// TIA Portal V16 export
// export: Created 2021-12-01T21:20:16.7242301Z, ExportSetting WithDefaults, DisplayName Totally Integrated Automation Portal, DisplayVersion V16 Update 4, DisplayName TIA Portal Version Control Interface, DisplayVersion V16 Update 2, DisplayName TIA Portal Openness, DisplayVersion V16 Update 4, DisplayName SINAMICS Startdrive Advanced, DisplayVersion V16 Update 5, DisplayName SINAMICS Startdrive G130, G150, S120, S150, SINAMICS MV, S210, DisplayVersion V16 Update 5, DisplayName SINAMICS Startdrive G110M, G120, G120C, G120D, G120P, G115D, DisplayVersion V16 Update 5, DisplayName STEP 7 Professional, DisplayVersion V16 Update 4, DisplayName STEP 7 Safety, DisplayVersion V16, DisplayName WinCC Advanced, DisplayVersion V16 Update 4
FUNCTION "ST00270_FC" : Void   // FC157, LAD
TITLE = ST00270
{ S7_Optimized_Access := 'TRUE' }
VERSION : 0.1
// stored: AutoNumber true, IsIECCheckEnabled false, SetENOAutomatically false, UDAEnableTagReadback false
   VAR_IN_OUT
      OPMODE : "OPMODE_OUT_UDT";
      HMI_EXTENSION : "HMI_EXTENSION_PANEL_UDT";
   END_VAR
BEGIN

REGION Network 1: Alarm
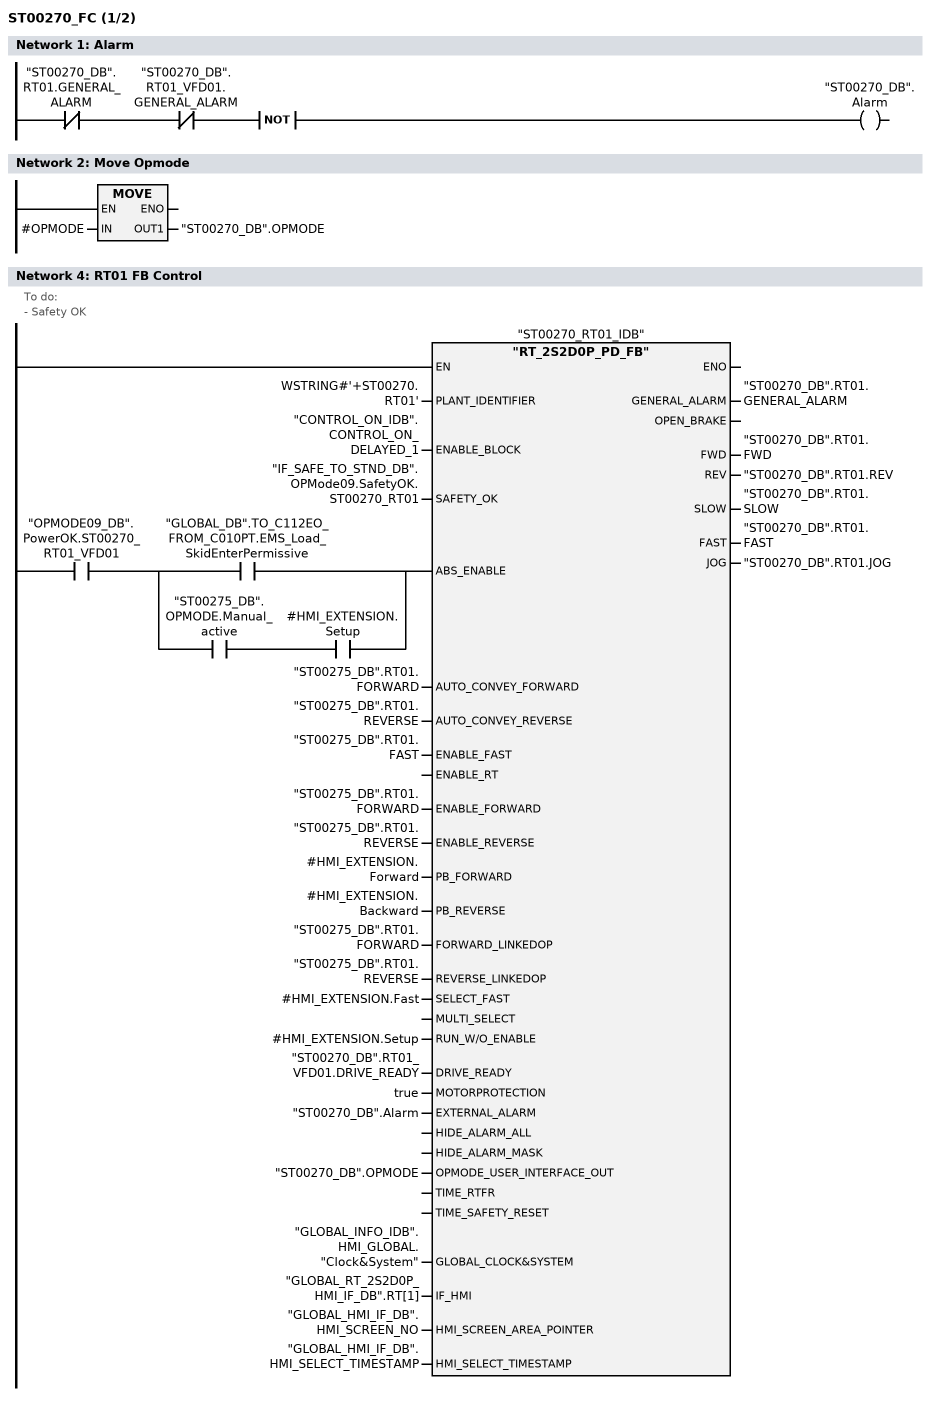
   RUNG wire#powerrail
      I_Contact( "ST00270_DB".RT01.GENERAL_ALARM )
      I_Contact( "ST00270_DB".RT01_VFD01.GENERAL_ALARM )
      Not()
      Coil( "ST00270_DB".Alarm )
   END_RUNG
   // the same network as SCL:
   "ST00270_DB".Alarm := NOT (NOT "ST00270_DB".RT01.GENERAL_ALARM AND NOT "ST00270_DB".RT01_VFD01.GENERAL_ALARM);
END_REGION

REGION Network 2: Move Opmode
   RUNG wire#powerrail
      Move(in := #OPMODE, out1 => "ST00270_DB".OPMODE)
   END_RUNG
   // the same network as SCL:
   "ST00270_DB".OPMODE := #OPMODE;
END_REGION

REGION Network 3: *******************RT01 Control*******************
END_REGION

REGION Network 4: RT01 FB Control
   // To do:
   // 										- Safety OK
   RUNG wire#powerrail
      "ST00270_RT01_IDB"(ABS_ENABLE := wire#w2, PLANT_IDENTIFIER := WSTRING#'+ST00270.RT01', ENABLE_BLOCK := "CONTROL_ON_IDB".CONTROL_ON_DELAYED_1, SAFETY_OK := "IF_SAFE_TO_STND_DB".OPMode09.SafetyOK.ST00270_RT01, AUTO_CONVEY_FORWARD := "ST00275_DB".RT01.FORWARD, AUTO_CONVEY_REVERSE := "ST00275_DB".RT01.REVERSE, ENABLE_FAST := "ST00275_DB".RT01.FAST, ENABLE_RT :=, ENABLE_FORWARD := "ST00275_DB".RT01.FORWARD, ENABLE_REVERSE := "ST00275_DB".RT01.REVERSE, PB_FORWARD := #HMI_EXTENSION.Forward, PB_REVERSE := #HMI_EXTENSION.Backward, FORWARD_LINKEDOP := "ST00275_DB".RT01.FORWARD, REVERSE_LINKEDOP := "ST00275_DB".RT01.REVERSE, SELECT_FAST := #HMI_EXTENSION.Fast, MULTI_SELECT :=, "RUN_W/O_ENABLE" := #HMI_EXTENSION.Setup, DRIVE_READY := "ST00270_DB".RT01_VFD01.DRIVE_READY, MOTORPROTECTION := true, EXTERNAL_ALARM := "ST00270_DB".Alarm, HIDE_ALARM_ALL :=, HIDE_ALARM_MASK :=, OPMODE_USER_INTERFACE_OUT := "ST00270_DB".OPMODE, TIME_RTFR :=, TIME_SAFETY_RESET :=, "GLOBAL_CLOCK&SYSTEM" := "GLOBAL_INFO_IDB".HMI_GLOBAL."Clock&System", IF_HMI := "GLOBAL_RT_2S2D0P_HMI_IF_DB".RT[1], HMI_SCREEN_AREA_POINTER := "GLOBAL_HMI_IF_DB".HMI_SCREEN_NO, HMI_SELECT_TIMESTAMP := "GLOBAL_HMI_IF_DB".HMI_SELECT_TIMESTAMP, GENERAL_ALARM => "ST00270_DB".RT01.GENERAL_ALARM, OPEN_BRAKE =>, FWD => "ST00270_DB".RT01.FWD, REV => "ST00270_DB".RT01.REV, SLOW => "ST00270_DB".RT01.SLOW, FAST => "ST00270_DB".RT01.FAST, JOG => "ST00270_DB".RT01.JOG)
   END_RUNG
   RUNG wire#powerrail
      Contact( "OPMODE09_DB".PowerOK.ST00270_RT01_VFD01 )
      wire#w1
      Contact( "GLOBAL_DB".TO_C112EO_FROM_C010PT.EMS_Load_SkidEnterPermissive )
   END_RUNG wire#w2
   RUNG wire#w1
      Contact( "ST00275_DB".OPMODE.Manual_active )
      Contact( #HMI_EXTENSION.Setup )
   END_RUNG wire#w2
   // the same network as SCL:
   "ST00270_RT01_IDB"(PLANT_IDENTIFIER := WSTRING#'+ST00270.RT01',   // "RT_2S2D0P_PD_FB"
                      ENABLE_BLOCK := "CONTROL_ON_IDB".CONTROL_ON_DELAYED_1,
                      SAFETY_OK := "IF_SAFE_TO_STND_DB".OPMode09.SafetyOK.ST00270_RT01,
                      ABS_ENABLE := "OPMODE09_DB".PowerOK.ST00270_RT01_VFD01 AND ("GLOBAL_DB".TO_C112EO_FROM_C010PT.EMS_Load_SkidEnterPermissive OR ("ST00275_DB".OPMODE.Manual_active AND #HMI_EXTENSION.Setup)),
                      AUTO_CONVEY_FORWARD := "ST00275_DB".RT01.FORWARD,
                      AUTO_CONVEY_REVERSE := "ST00275_DB".RT01.REVERSE,
                      ENABLE_FAST := "ST00275_DB".RT01.FAST,
                      ENABLE_FORWARD := "ST00275_DB".RT01.FORWARD,
                      ENABLE_REVERSE := "ST00275_DB".RT01.REVERSE,
                      PB_FORWARD := #HMI_EXTENSION.Forward,
                      PB_REVERSE := #HMI_EXTENSION.Backward,
                      FORWARD_LINKEDOP := "ST00275_DB".RT01.FORWARD,
                      REVERSE_LINKEDOP := "ST00275_DB".RT01.REVERSE,
                      SELECT_FAST := #HMI_EXTENSION.Fast,
                      "RUN_W/O_ENABLE" := #HMI_EXTENSION.Setup,
                      DRIVE_READY := "ST00270_DB".RT01_VFD01.DRIVE_READY,
                      MOTORPROTECTION := true,
                      EXTERNAL_ALARM := "ST00270_DB".Alarm,
                      OPMODE_USER_INTERFACE_OUT := "ST00270_DB".OPMODE,
                      "GLOBAL_CLOCK&SYSTEM" := "GLOBAL_INFO_IDB".HMI_GLOBAL."Clock&System",
                      IF_HMI := "GLOBAL_RT_2S2D0P_HMI_IF_DB".RT[1],
                      HMI_SCREEN_AREA_POINTER := "GLOBAL_HMI_IF_DB".HMI_SCREEN_NO,
                      HMI_SELECT_TIMESTAMP := "GLOBAL_HMI_IF_DB".HMI_SELECT_TIMESTAMP,
                      GENERAL_ALARM => "ST00270_DB".RT01.GENERAL_ALARM,
                      FWD => "ST00270_DB".RT01.FWD,
                      REV => "ST00270_DB".RT01.REV,
                      SLOW => "ST00270_DB".RT01.SLOW,
                      FAST => "ST00270_DB".RT01.FAST,
                      JOG => "ST00270_DB".RT01.JOG);
END_REGION

REGION Network 5: RT01 Speed
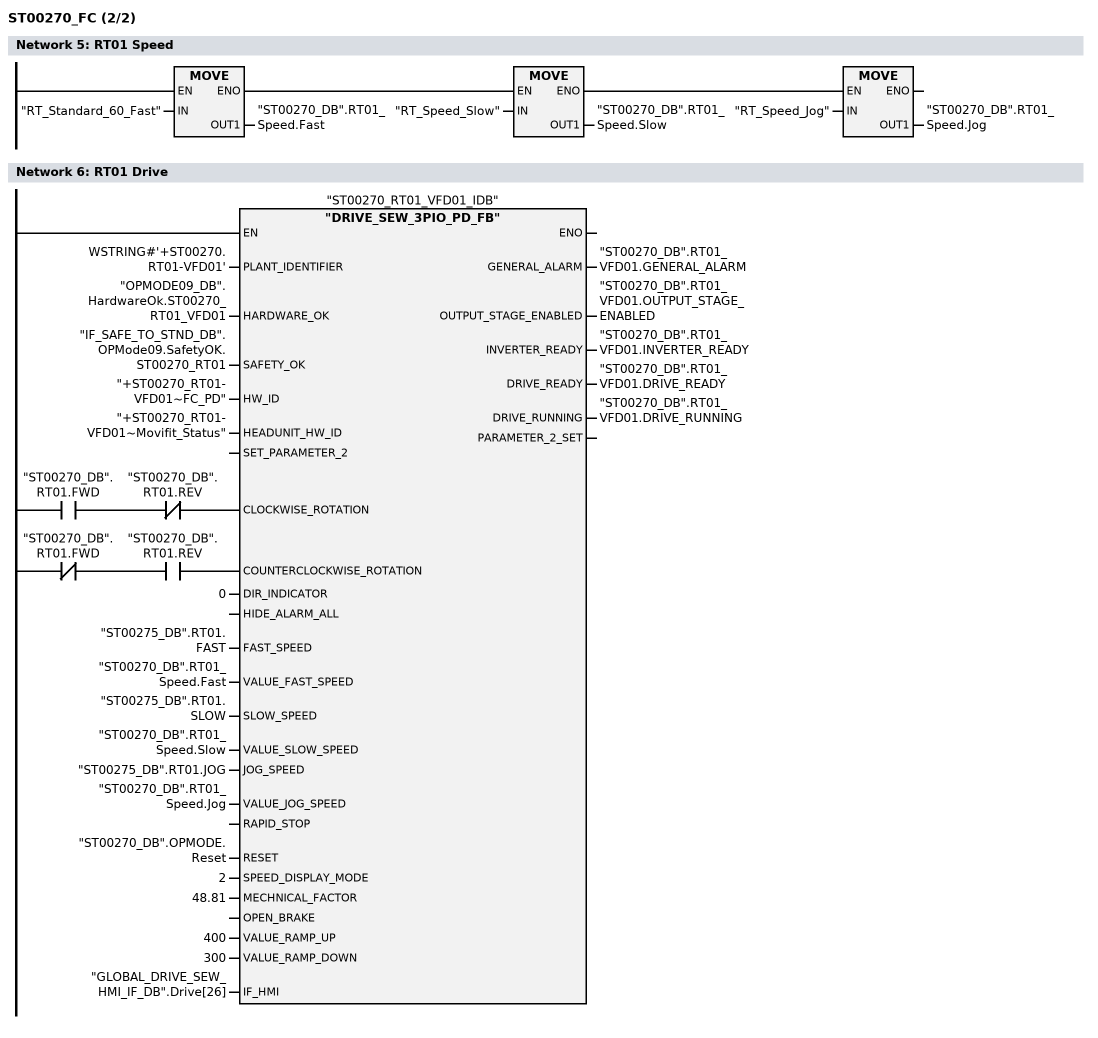
   RUNG wire#powerrail
      Move(in := "RT_Standard_60_Fast", out1 => "ST00270_DB".RT01_Speed.Fast)
      Move(in := "RT_Speed_Slow", out1 => "ST00270_DB".RT01_Speed.Slow)
      Move(in := "RT_Speed_Jog", out1 => "ST00270_DB".RT01_Speed.Jog)
   END_RUNG
   // the same network as SCL:
   "ST00270_DB".RT01_Speed.Fast := "RT_Standard_60_Fast";
   "ST00270_DB".RT01_Speed.Slow := "RT_Speed_Slow";
   "ST00270_DB".RT01_Speed.Jog := "RT_Speed_Jog";
END_REGION

REGION Network 6: RT01 Drive
   RUNG wire#powerrail
      "ST00270_RT01_VFD01_IDB"(CLOCKWISE_ROTATION := wire#w1, COUNTERCLOCKWISE_ROTATION := wire#w2, PLANT_IDENTIFIER := WSTRING#'+ST00270.RT01-VFD01', HARDWARE_OK := "OPMODE09_DB".HardwareOk.ST00270_RT01_VFD01, SAFETY_OK := "IF_SAFE_TO_STND_DB".OPMode09.SafetyOK.ST00270_RT01, HW_ID := "+ST00270_RT01-VFD01~FC_PD", HEADUNIT_HW_ID := "+ST00270_RT01-VFD01~Movifit_Status", SET_PARAMETER_2 :=, DIR_INDICATOR := 0, HIDE_ALARM_ALL :=, FAST_SPEED := "ST00275_DB".RT01.FAST, VALUE_FAST_SPEED := "ST00270_DB".RT01_Speed.Fast, SLOW_SPEED := "ST00275_DB".RT01.SLOW, VALUE_SLOW_SPEED := "ST00270_DB".RT01_Speed.Slow, JOG_SPEED := "ST00275_DB".RT01.JOG, VALUE_JOG_SPEED := "ST00270_DB".RT01_Speed.Jog, RAPID_STOP :=, RESET := "ST00270_DB".OPMODE.Reset, SPEED_DISPLAY_MODE := 2, MECHNICAL_FACTOR := 48.81, OPEN_BRAKE :=, VALUE_RAMP_UP := 400, VALUE_RAMP_DOWN := 300, IF_HMI := "GLOBAL_DRIVE_SEW_HMI_IF_DB".Drive[26], GENERAL_ALARM => "ST00270_DB".RT01_VFD01.GENERAL_ALARM, OUTPUT_STAGE_ENABLED => "ST00270_DB".RT01_VFD01.OUTPUT_STAGE_ENABLED, INVERTER_READY => "ST00270_DB".RT01_VFD01.INVERTER_READY, DRIVE_READY => "ST00270_DB".RT01_VFD01.DRIVE_READY, DRIVE_RUNNING => "ST00270_DB".RT01_VFD01.DRIVE_RUNNING, PARAMETER_2_SET =>)
   END_RUNG
   RUNG wire#powerrail
      Contact( "ST00270_DB".RT01.FWD )
      I_Contact( "ST00270_DB".RT01.REV )
   END_RUNG wire#w1
   RUNG wire#powerrail
      I_Contact( "ST00270_DB".RT01.FWD )
      Contact( "ST00270_DB".RT01.REV )
   END_RUNG wire#w2
   // the same network as SCL:
   "ST00270_RT01_VFD01_IDB"(PLANT_IDENTIFIER := WSTRING#'+ST00270.RT01-VFD01',   // "DRIVE_SEW_3PIO_PD_FB"
                           HARDWARE_OK := "OPMODE09_DB".HardwareOk.ST00270_RT01_VFD01,
                           SAFETY_OK := "IF_SAFE_TO_STND_DB".OPMode09.SafetyOK.ST00270_RT01,
                           HW_ID := "+ST00270_RT01-VFD01~FC_PD",
                           HEADUNIT_HW_ID := "+ST00270_RT01-VFD01~Movifit_Status",
                           CLOCKWISE_ROTATION := "ST00270_DB".RT01.FWD AND NOT "ST00270_DB".RT01.REV,
                           COUNTERCLOCKWISE_ROTATION := NOT "ST00270_DB".RT01.FWD AND "ST00270_DB".RT01.REV,
                           DIR_INDICATOR := 0,
                           FAST_SPEED := "ST00275_DB".RT01.FAST,
                           VALUE_FAST_SPEED := "ST00270_DB".RT01_Speed.Fast,
                           SLOW_SPEED := "ST00275_DB".RT01.SLOW,
                           VALUE_SLOW_SPEED := "ST00270_DB".RT01_Speed.Slow,
                           JOG_SPEED := "ST00275_DB".RT01.JOG,
                           VALUE_JOG_SPEED := "ST00270_DB".RT01_Speed.Jog,
                           RESET := "ST00270_DB".OPMODE.Reset,
                           SPEED_DISPLAY_MODE := 2,
                           MECHNICAL_FACTOR := 48.81,
                           VALUE_RAMP_UP := 400,
                           VALUE_RAMP_DOWN := 300,
                           IF_HMI := "GLOBAL_DRIVE_SEW_HMI_IF_DB".Drive[26],
                           GENERAL_ALARM => "ST00270_DB".RT01_VFD01.GENERAL_ALARM,
                           OUTPUT_STAGE_ENABLED => "ST00270_DB".RT01_VFD01.OUTPUT_STAGE_ENABLED,
                           INVERTER_READY => "ST00270_DB".RT01_VFD01.INVERTER_READY,
                           DRIVE_READY => "ST00270_DB".RT01_VFD01.DRIVE_READY,
                           DRIVE_RUNNING => "ST00270_DB".RT01_VFD01.DRIVE_RUNNING);
END_REGION
END_FUNCTION
